FUNCTION_BLOCK RunningToHaltedUnifiedProgramTransition EXTENDS RunningToHaltedProgramTransition
VAR_STAT
	//! <summary>Class name shared by all instances of this function block.</summary>
	{attribute 'OPC.UA.DA' := '0'}
	_ClassName : STRING := __POUNAME();
END_VAR

{attribute 'monitoring' := 'call'}
PROPERTY ClassName : REFERENCE TO STRING
GET
ClassName REF= _ClassName;
END_GET
END_PROPERTY

END_FUNCTION_BLOCK

(* stored: Version 1.1.0.1
   POU RunningToHaltedUnifiedProgramTransition: Id {cc26bbc4-9747-4e71-9ca8-bd1f63556de1}, SpecialFunc None
   Property ClassName: Id {8050dc7d-7927-4886-95ff-fbd15437b979}
   Get Get: Id {5d5055e5-b23d-4a48-80ec-80537befc11b} *)
